{attribute 'no_explicit_call' := 'do not call this function block directly'} 
FUNCTION_BLOCK DeleteDirectory EXTENDS ToolkitObject IMPLEMENTS IAction
VAR
	{attribute 'OPC.UA.DA' := '0'}
	_ClassName : STRING := __POUNAME();

	{attribute 'OPC.UA.DA' := '0'}
    _DeleteDirectory : Tc2_System.FB_RemoveDir;	
	
	{attribute 'OPC.UA.DA' := '0'}
	_NeedStart : BOOL;
	{attribute 'OPC.UA.DA' := '0'}
	_Done : BOOL;
END_VAR

{attribute 'monitoring' := 'call'}
{attribute 'OPC.UA.DA.Property' := '1'}
{attribute 'OPC.UA.DA' := '1'}
PROPERTY AmsNetId : Tc2_System.T_AmsNetID
GET
AmsNetId := _DeleteDirectory.sNetId;
END_GET
SET
_DeleteDirectory.sNetId := AmsNetId;
END_SET
END_PROPERTY

{attribute 'monitoring' := 'call'}
{attribute 'OPC.UA.DA.Property' := '1'}
{attribute 'OPC.UA.DA.Access' := '1'}
PROPERTY Busy : BOOL
GET
Busy := _NeedStart OR_ELSE _DeleteDirectory.bBusy;
END_GET
END_PROPERTY

{attribute 'monitoring' := 'call'}
PROPERTY ClassName : STRING
GET
ClassName := _ClassName;
END_GET
END_PROPERTY

{attribute 'monitoring' := 'call'}
{attribute 'OPC.UA.DA.Property' := '1'}
{attribute 'OPC.UA.DA.Access' := '1'}
PROPERTY Done : BOOL
GET
Done := _Done;
END_GET
END_PROPERTY

{attribute 'monitoring' := 'call'}
{attribute 'OPC.UA.DA.Property' := '1'}
{attribute 'OPC.UA.DA.Access' := '1'}
PROPERTY Error : BOOL
GET
Error := _DeleteDirectory.bError;
END_GET
END_PROPERTY

METHOD Execute
VAR
	errorMessage : ERROR_MESSAGE;
END_VAR
IF _NeedStart OR_ELSE _DeleteDirectory.bBusy THEN
	_DeleteDirectory(bExecute := TRUE);
	_NeedStart := FALSE;
	
	IF _DeleteDirectory.bError THEN
		errorMessage := "An error occurred while deleting the directory '";
		WStringHelper.Append2(errorMessage, TO_WSTRING(_DeleteDirectory.sPathName), "'");	
		_LastException.Configure(errorMessage, __POUNAME(), ClassName, CurrentNamespace.Name, __POSITION(), _DeleteDirectory.nErrId).Throw();
	ELSIF NOT _DeleteDirectory.bBusy THEN
		_Done := TRUE;
	END_IF
END_IF
END_METHOD

{attribute 'monitoring' := 'call'}
{attribute 'OPC.UA.DA.Property' := '1'}
{attribute 'OPC.UA.DA.Access' := '1'}
PROPERTY LastException : REFERENCE TO Exception
GET
LastException REF= _LastException;
END_GET
END_PROPERTY

{attribute 'monitoring' := 'call'}
{attribute 'OPC.UA.DA.Property' := '1'}
{attribute 'OPC.UA.DA' := '1'}
PROPERTY PathType : Tc2_System.E_OpenPath
GET
PathType := _DeleteDirectory.ePath;
END_GET
SET
_DeleteDirectory.ePath := PathType;
END_SET
END_PROPERTY

METHOD Start
VAR_INPUT
	directoryPath : Tc2_System.T_MaxString;
END_VAR
_NeedStart := TRUE;
_Done := FALSE;
_DeleteDirectory.sPathName := directoryPath;

_LastException.Clear();
END_METHOD

{attribute 'monitoring' := 'call'}
{attribute 'OPC.UA.DA.Property' := '1'}
{attribute 'OPC.UA.DA' := '1'}
PROPERTY Timeout : TIME
GET
Timeout := _DeleteDirectory.tTimeout;
END_GET
SET
_DeleteDirectory.tTimeout := Timeout;
END_SET
END_PROPERTY

END_FUNCTION_BLOCK

(* stored: Version 1.1.0.1
   POU DeleteDirectory: Id {ddf25607-39dd-4f09-9865-1a874e7acdd3}, SpecialFunc None
   Property AmsNetId: Id {9a3b6a1b-903b-47b7-88cf-aad9420711db}
   Get Get: Id {a25ce6d9-968d-4bd1-be9d-06706c5bb275}
   Set Set: Id {f23eede0-3454-4176-8028-823c80082567}
   Property Busy: Id {30449498-9c29-4af0-8abe-a82c31d0af6e}
   Get Get: Id {7b41b589-2291-471c-8743-242785cb1508}
   Property ClassName: Id {c382225d-773e-44b0-9ac6-4b83fb2e6e39}
   Get Get: Id {b8920e5a-6746-40df-81bd-2ddb536aa132}
   Property Done: Id {8e374970-c733-4564-b133-060b033611f2}
   Get Get: Id {bfd7b12a-ffa9-498d-8046-aeeaa64f5174}
   Property Error: Id {fcc495f4-12c8-4953-8fb2-65e146de84ba}
   Get Get: Id {54b8758b-43ee-4ce6-9d42-0f6822e4ba77}
   Method Execute: Id {5721afc5-c2c4-4aeb-98cc-6f3e84343944}
   Property LastException: Id {fc1716af-fa7f-46c8-94ec-a5e5648b3848}
   Get Get: Id {a811c779-9d20-401a-b0aa-b7475130a415}
   Property PathType: Id {b245c4fa-fde4-4b85-b852-4369f35419af}
   Get Get: Id {1cc7560f-b75a-4f6a-aa0f-415f02f8ee96}
   Set Set: Id {3ee60c5b-532e-4ebe-9010-e3011d6903fb}
   Method Start: Id {82534506-7cea-4bec-b625-96c2722965db}
   Property Timeout: Id {92a72712-830b-4e13-aa58-9cd8af105736}
   Get Get: Id {43eca328-995e-455a-98a3-bad372537338}
   Set Set: Id {524a0066-8913-49a5-92bb-ec9f677f7a24} *)
